FUNCTION_BLOCK TCTR_Logic (* Basic Function Block Type *)
  (* Standard: 61499-2 *)
  (* Version 0.0, 12/10/2023, Cheyan, Schneider Electric, Template *)
  PACKAGE Main;
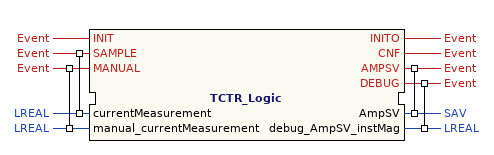
  EVENT_INPUT
    INIT; (* Initialization Request *)
    SAMPLE WITH currentMeasurement; (* Normal Execution Request *)
    MANUAL WITH manual_currentMeasurement;
  END_EVENT
  EVENT_OUTPUT
    INITO; (* Initialization Confirm *)
    CNF; (* Execution Confirmation *)
    AMPSV WITH AmpSV;
    DEBUG WITH debug_AmpSV_instMag;
  END_EVENT
  VAR_INPUT
    currentMeasurement : LREAL; (* Input event qualifier *)
    manual_currentMeasurement : LREAL;
  END_VAR
  VAR_OUTPUT
    AmpSV : SAV; (* Output event qualifier *)
    debug_AmpSV_instMag : LREAL;
  END_VAR
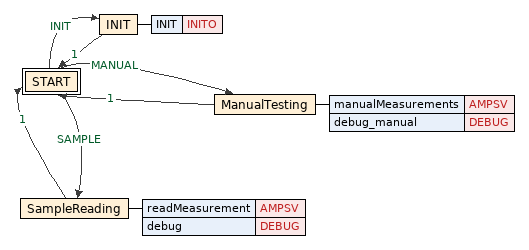
  EC_STATES
    START; (* Initial State *)
    INIT : INIT -> INITO; (* Initialization *)
    SampleReading : readMeasurement -> AMPSV, debug -> DEBUG; (* Normal execution *)
    ManualTesting : manualMeasurements -> AMPSV, debug_manual -> DEBUG;
  END_STATES
  EC_TRANSITIONS
    START TO INIT := INIT;
    INIT TO START := 1;
    START TO SampleReading := SAMPLE;
    SampleReading TO START := 1;
    START TO ManualTesting := MANUAL;
    ManualTesting TO START := 1;
  END_TRANSITIONS
  ALGORITHM INIT IN ST: (* Initialization algorithm *)
;
  END_ALGORITHM
  ALGORITHM readMeasurement IN ST: (* Normally executed algorithm The analogue measurement from the electrical system (plant) is digitalized to an IEC61850 variable *)
;

AmpSV.instMag.f := currentMeasurement;
  END_ALGORITHM
  ALGORITHM debug IN ST: (* Debugging *)
;

debug_AmpSV_instMag := currentMeasurement;
  END_ALGORITHM
  ALGORITHM manualMeasurements IN ST:
;

AmpSV.instMag.f := manual_currentMeasurement;
  END_ALGORITHM
  ALGORITHM debug_manual IN ST:
;

debug_AmpSV_instMag := manual_currentMeasurement;
  END_ALGORITHM
END_FUNCTION_BLOCK
